TYPE ST_SafetyFunctionOut :
STRUCT
    bDiagOk: BIT; //OK (Where diagnostics need TO be checked, i.e. drive errors)
    bOutput: BIT; //Where PLC checks consistency (i.e. STO)
    bRequest: BIT;
    bDummy: BIT; //Not in use
END_STRUCT
END_TYPE

(* stored: Version 1.1.0.1
   DUT ST_SafetyFunctionOut: Id {d225f0e9-f4be-0268-2036-d232ca0275b9} *)
